# EPICS autosave request: medipixApp/Db/medipix_settings.req
file "ADBase_settings.req" P=$(P), R=$(R)
$(P)$(R)QuadMerlinMode
$(P)$(R)OperatingEnergy
$(P)$(R)ThresholdEnergy0
$(P)$(R)ThresholdEnergy1
$(P)$(R)ThresholdEnergy2
$(P)$(R)ThresholdEnergy3
$(P)$(R)ThresholdEnergy4
$(P)$(R)ThresholdEnergy5
$(P)$(R)ThresholdEnergy6
$(P)$(R)ThresholdEnergy7
$(P)$(R)ThresholdScan
$(P)$(R)StartThresholdScan
$(P)$(R)StopThresholdScan
$(P)$(R)StepThresholdScan
